// TIA Portal V17 export
// export: Created 2023-02-13T11:16:11.2408746Z, ExportSetting WithDefaults, DisplayName Totally Integrated Automation Portal, DisplayVersion V17, DisplayName TIA Portal Openness, DisplayVersion V17, DisplayName TIA Portal Teamcenter Gateway, DisplayVersion V17, DisplayName TIA Portal Version Control Interface, DisplayVersion V17, DisplayName SINAMICS Startdrive Advanced, DisplayVersion V17, DisplayName SINAMICS Startdrive G130, G150, S120, S150, SINAMICS MV, S210, DisplayVersion V17, DisplayName SINAMICS Startdrive G110M, G120, G120C, G120D, G120P, G115D, DisplayVersion V17, DisplayName STEP 7 Professional, DisplayVersion V17, DisplayName STEP 7 Safety, DisplayVersion V17, DisplayName WinCC Professional, DisplayVersion V17
DATA_BLOCK "Blend_T-31"   // DB214
VERSION : 0.1
// stored: AutoNumber false, DBAccessibleFromOPCUA true, DBAccessibleFromWebserver true, InstanceOfName Blend_Tank, InstanceOfType FB
"Blend_Tank"
   // VAR_INPUT
   //    IN_FBAV_Header1 : Bool;
   //    IN_FBAV_Header2 : Bool;
   //    IN_FBAV_Vinegar : Bool;
   //    IN_FBAV_Sugar : Bool;
   //    IN_FBAV_Salt : Bool;
   //    IN_FBAV_ProWater : Bool;
   //    IN_FBAV_Homomixer : Bool;
   //    IN_FBAV_Transfer1 : Bool;
   //    IN_FBAV_Transfer2 : Bool;
   //    IN_FBAV_Transfer3 : Bool;
   //    IN_FBAV_Outlet : Bool;
   //    IN_FBAV_CIP : Bool;
   //    IN_FBP_Transfer1 : Bool;
   //    IN_FBP_Transfer1_Sp : Real;
   //    IN_FBP_Transfer2 : Bool;
   //    IN_FBP_Transfer2_Sp : Real;
   //    IN_FBP_Transfer3 : Bool;
   //    IN_FBP_Transfer3_Sp : Real;
   //    IN_FBP_CIP : Bool;
   //    IN_FBP_CIP_Sp : Real;
   //    IN_LT01 : Real;
   //    "BFT-1 Prod Req" : Bool;
   //    "BFT-1 Prod Line" : Bool;
   //    "BFT-1 CIP Enable" : Bool;
   //    "BFT-1 CIPLine" : Bool;
   //    "BFT-2 Prod Req" : Bool;
   //    "BFT-2 Prod Line" : Bool;
   //    "BFT-2 CIP Enable" : Bool;
   //    "BFT-2 CIPLine" : Bool;
   //    "BFT-3 Prod Req" : Bool;
   //    "BFT-3 Prod Line" : Bool;
   //    "BFT-3 CIP Enable" : Bool;
   //    "BFT-3 CIPLine" : Bool;
   //    "Transfer 1 Busy" : Bool;
   //    "Transfer 2 Busy" : Bool;
   //    "Transfer 3 Busy" : Bool;
   //    "Header 1 Available" : Bool;
   //    "Header 2 Available" : Bool;
   //    "Vinegar Available" : Bool;
   //    "Sugar Available" : Bool;
   //    "Salt Available" : Bool;
   //    "ProWater Available" : Bool;
   //    "Homomixer Available" : Bool;
   //    IN_LDT : Date_And_Time;
   //    "CIP Pulse" : Bool;
   //    "CIP Supply ON" : Bool;
   //    "CIP Req OK" : Bool;
   //    "CIP Complete" : Bool;
   //    "CIP Busy" : Bool;
   // END_VAR
   // VAR_OUTPUT
   //    Out_AV_Header1 : Bool;
   //    Out_AV_Header2 : Bool;
   //    Out_AV_Vinegar : Bool;
   //    Out_AV_Sugar : Bool;
   //    Out_AV_Salt : Bool;
   //    Out_AV_ProWater : Bool;
   //    Out_AV_Homomixer : Bool;
   //    Out_AV_Transfer1 : Bool;
   //    Out_AV_Transfer2 : Bool;
   //    Out_AV_Transfer3 : Bool;
   //    Out_AV_Outlet : Bool;
   //    Out_AV_CIP : Bool;
   //    Out_P_Transfer1 : Bool;
   //    Out_P_Transfer1_Sp : Real;
   //    Out_P_Transfer2 : Bool;
   //    Out_P_Transfer2_Sp : Real;
   //    Out_P_Transfer3 : Bool;
   //    Out_P_Transfer3_Sp : Real;
   //    Out_P_CIP : Bool;
   //    Out_P_CIP_Sp : Real;
   //    Out_Agi : Bool;
   //    Out_Agi_Sp : Real;
   //    "Header 1 Req" : Bool;
   //    "Header 2 Req" : Bool;
   //    "Vinegar Req" : Bool;
   //    "Sugar Req" : Bool;
   //    "Salt Req" : Bool;
   //    "ProWater Req" : Bool;
   //    "Homomixer Req" : Bool;
   //    Out_CIP_Req : Bool;
   //    Out_CIP_Line_Open : Bool;
   // END_VAR
   // VAR
   //    Cmd : Struct
   //       "Ready For Transfer" : Bool;
   //       "CIP Tank 1" : Bool;
   //       "CIP Tank 2" : Bool;
   //       "CIP Line" : Bool;
   //       "Dose Head 1" : Bool;
   //       "Dose Head 2" : Bool;
   //       Agitator_Mode : Bool;
   //    END_STRUCT;
   // END_VAR
   // VAR RETAIN
   //    Param : Struct
   //       SP_Level_LL : Real;
   //       SP_Level_ML : Real;
   //       SP_Level_HL : Real;
   //       L_Hi_Lim : Real;
   //       L_Lo_Lim : Real;
   //       L_Hys : Real;
   //       LB_ON : Real;
   //       LB_OFF : Real;
   //       LB1_ON : Real;
   //       LB1_OFF : Real;
   //       LB2_ON : Real;
   //       LB2_OFF : Real;
   //       LB3_ON : Real;
   //       LB3_OFF : Real;
   //       SP_P1_Speed : Real;
   //       SP_P2_Speed : Real;
   //       SP_P3_Speed : Real;
   //       SP_LB_Speed : Real;
   //       SP_LB1_Speed : Real;
   //       SP_LB2_Speed : Real;
   //       SP_LB3_Speed : Real;
   //       CIP_Tank_P_Ret_Speed : Real;
   //       CIP_Ret_ON_SP : Real;
   //       CIP_Ret_OFF_SP : Real;
   //       Flushing_HW_Timer : Time;
   //    END_STRUCT;
   // END_VAR
   // VAR
   //    State : Struct
   //       "Tank LL" : Bool;
   //       "Tank ML" : Bool;
   //       "Tank HL" : Bool;
   //       LB_ON : Bool;
   //       LB1_ON : Bool;
   //       LB2_ON : Bool;
   //       LB3_ON : Bool;
   //       "CIP Tank" : Bool;
   //       "CIP Tank Ena" : Bool;
   //       "CIP Tank Ret 1 Ena" : Bool;
   //       "CIP Tank Ret 2 Ena" : Bool;
   //       "CIP Line" : Bool;
   //       "CIP Line Ena" : Bool;
   //       "CIP Return On" : Bool;
   //       "Dose On Prog" : Bool;
   //       "Dose EN" : Bool;
   //       "Ready For Transfer" : Bool;
   //       "Ready For Transfer Ena" : Bool;
   //       "BFT-1 EN" : Bool;
   //       "BFT-2 EN" : Bool;
   //       "BFT-3 EN" : Bool;
   //       "RM Dose" : Bool;
   //       "Transfer 1 On Progress" : Bool;
   //       "Transfer 2 On Progress" : Bool;
   //       "Transfer 3 On Progress" : Bool;
   //       "DoseHead1 ON" : Bool;
   //       "DoseHead2 ON" : Bool;
   //    END_STRUCT;
   //    Dose : Struct
   //       Dose_Start : DWord;
   //       Dose_Pause : DWord;
   //       Dose_Stop : DWord;
   //       Dose_State : DWord;
   //       Dose_Tank_Available : Word;
   //       Dose_Prod_Ready : Word;
   //       Dose_Header_Req : DWord;
   //       Dose_EN : Word;
   //    END_STRUCT;
   //    "Dose_Level_%" : Struct
   //       "ChiliAwetan1%" : Real;
   //       "ChiliAwetan2%" : Real;
   //       "ChiliAwetan3%" : Real;
   //       "Tomato%" : Real;
   //       "ChiliFresh1%" : Real;
   //       "ChiliFresh2%" : Real;
   //       "ChiliFresh3%" : Real;
   //       "Garlic%" : Real;
   //       "HW%" : Real;
   //       "Vinegar%" : Real;
   //       "Sugar%" : Real;
   //       "Salt%" : Real;
   //       "ProWater%" : Real;
   //       "Homomixer%" : Real;
   //    END_STRUCT;
   //    Dose_Level_Lit : Struct
   //       ChiliAwetan1Lit : Real;
   //       ChiliAwetan2Lit : Real;
   //       ChiliAwetan3Lit : Real;
   //       TomatoLit : Real;
   //       ChiliFresh1Lit : Real;
   //       ChiliFresh2Lit : Real;
   //       ChiliFresh3Lit : Real;
   //       GarlicLit : Real;
   //       HWLit : Real;
   //       VinegarLit : Real;
   //       SugarLit : Real;
   //       SaltLit : Real;
   //       ProWaterLit : Real;
   //       HomomixerLit : Real;
   //    END_STRUCT;
   //    SP_Dose_Level : Struct
   //       ChiliAwetan1Lit : Real;
   //       ChiliAwetan2Lit : Real;
   //       ChiliAwetan3Lit : Real;
   //       TomatoLit : Real;
   //       ChiliFresh1Lit : Real;
   //       ChiliFresh2Lit : Real;
   //       ChiliFresh3Lit : Real;
   //       GarlicLit : Real;
   //       HWLit : Real;
   //       VinegarLit : Real;
   //       SugarLit : Real;
   //       SaltLit : Real;
   //       ProWaterLit : Real;
   //       HomomixerLit : Real;
   //    END_STRUCT;
   //    r : Struct
   //       PosE1 : Bool;
   //       PosE2 : Bool;
   //       PosE3 : Bool;
   //       PosE4 : Bool;
   //       PosE5 : Bool;
   //       PosE6 : Bool;
   //       PosE7 : Bool;
   //       PosE8 : Bool;
   //       PosE9 : Bool;
   //       PosE10 : Bool;
   //       PosE11 : Bool;
   //       PosE12 : Bool;
   //       PosE13 : Bool;
   //       PosE14 : Bool;
   //       PosE15 : Bool;
   //       PosE16 : Bool;
   //       PosE17 : Bool;
   //       PosE18 : Bool;
   //       PosE19 : Bool;
   //       PosE20 : Bool;
   //       PosE21 : Bool;
   //       PosE22 : Bool;
   //       PosE23 : Bool;
   //       PosE24 : Bool;
   //       PosE25 : Bool;
   //       PosE26 : Bool;
   //       PosE27 : Bool;
   //       PosE28 : Bool;
   //       PosE29 : Bool;
   //       PosE30 : Bool;
   //       PosE31 : Bool;
   //       PosE32 : Bool;
   //    END_STRUCT;
   //    Actuator : Struct
   //       P_Transfer1 : Bool;
   //       P_Transfer2 : Bool;
   //       P_Transfer3 : Bool;
   //       AV_Transfer1 : Bool;
   //       AV_Transfer2 : Bool;
   //       AV_Transfer3 : Bool;
   //       AV_Outlet : Bool;
   //       AV_CIP_Tank : Bool;
   //    END_STRUCT;
   //    SP_ChiliAwetan1 : "RawDose";
   //    SP_ChiliAwetan2 : "RawDose";
   //    SP_ChiliAwetan3 : "RawDose";
   //    SP_Tomato : "RawDose";
   //    SP_ChiliFresh1 : "RawDose";
   //    SP_ChiliFresh2 : "RawDose";
   //    SP_ChiliFresh3 : "RawDose";
   //    SP_Garlic : "RawDose";
   //    SP_HW : "Raw_Pulse";
   //    SP_Vinegar : "RawDose";
   //    SP_Sugar : "RawDose";
   //    SP_Salt : "RawDose";
   //    SP_ProWater : "Raw_Pulse";
   //    SP_Homomixer : "RawDose";
   //    Dose_ChiliAwetan1 { S7_SetPoint := 'True'} : "DOSE";
   //    Dose_ChiliAwetan2 { S7_SetPoint := 'True'} : "DOSE";
   //    Dose_ChiliAwetan3 { S7_SetPoint := 'True'} : "DOSE";
   //    Dose_Tomato { S7_SetPoint := 'True'} : "DOSE";
   //    Dose_ChiliFresh1 { S7_SetPoint := 'True'} : "DOSE";
   //    Dose_ChiliFresh2 { S7_SetPoint := 'True'} : "DOSE";
   //    Dose_ChiliFresh3 { S7_SetPoint := 'True'} : "DOSE";
   //    Dose_Garlic { S7_SetPoint := 'True'} : "DOSE";
   //    Dose_HW { S7_SetPoint := 'True'} : "DOSE";
   //    Dose_Vinegar { S7_SetPoint := 'True'} : "DOSE";
   //    Dose_Sugar { S7_SetPoint := 'True'} : "DOSE";
   //    Dose_Salt { S7_SetPoint := 'True'} : "DOSE";
   //    Dose_ProWater { S7_SetPoint := 'True'} : "DOSE";
   //    Dose_Homomixer { S7_SetPoint := 'True'} : "DOSE";
   //    AlwaysON { S7_SetPoint := 'True'} : Bool;
   //    L_Hys_Abs { S7_SetPoint := 'True'} : Real;
   //    Hys_Level_HL : Real;
   //    Hys_Level_ML : Real;
   //    Hys_Level_LL : Real;
   //    TimerOff_Valve_Out : TON_TIME;
   //    TimerOff_Valve_P_1 { S7_SetPoint := 'True'} : TON_TIME;
   //    TimerOff_Valve_P_2 { S7_SetPoint := 'True'} : TON_TIME;
   //    TimerOff_Valve_P_3 { S7_SetPoint := 'True'} : TON_TIME;
   //    TimerOff_Valve_P_CIP { S7_SetPoint := 'True'} : TON_TIME;
   // END_VAR
   // VAR RETAIN
   //    Last_Dose_Qty : Struct
   //       ChiliAwetan1 : Real;
   //       ChiliAwetan2 : Real;
   //       ChiliAwetan3 : Real;
   //       Tomato : Real;
   //       ChiliFresh1 : Real;
   //       ChiliFresh2 : Real;
   //       ChiliFresh3 : Real;
   //       Garlic : Real;
   //       HW : Real;
   //       Vinegar : Real;
   //       Sugar : Real;
   //       Salt : Real;
   //       ProWater : Real;
   //       Homomixer : Real;
   //    END_STRUCT;
   // END_VAR
   // VAR
   //    "HW Flushing" : Struct
   //       Status : Struct
   //          "Flush to Blend" : Bool;
   //          "Flush to Drain" : Bool;
   //          Drain : Bool;
   //          Done : Bool;
   //       END_STRUCT;
   //       Qty : Struct
   //          "Flush to Blend Qty" : Real;
   //          "Flush to Drain Qty" : Real;
   //          "Flush to Blend Act" : Real;
   //          "Flush to Drain Act" : Real;
   //       END_STRUCT;
   //       TimeDrain_SP : DInt;
   //       Cmd_Start_Drain : Bool;
   //       Cmd_Stop_Drain : Bool;
   //       DrainTime : TONR_TIME;
   //    END_STRUCT;
   //    PumpTF1_OnDelay : TON_TIME;
   //    PumpTF2_OnDelay { S7_SetPoint := 'True'} : TON_TIME;
   //    PumpTF3_OnDelay { S7_SetPoint := 'True'} : TON_TIME;
   // END_VAR
   // VAR RETAIN
   //    TimerON : Struct
   //       TimerON_1 : TON_TIME;
   //       TimerON_2 { S7_SetPoint := 'True'} : TON_TIME;
   //       TimerON_3 { S7_SetPoint := 'True'} : TON_TIME;
   //       TimerON_4 { S7_SetPoint := 'True'} : TON_TIME;
   //       TimerON_5 { S7_SetPoint := 'True'} : TON_TIME;
   //       TimerON_6 { S7_SetPoint := 'True'} : TON_TIME;
   //       TimerON_7 { S7_SetPoint := 'True'} : TON_TIME;
   //       TimerON_8 { S7_SetPoint := 'True'} : TON_TIME;
   //    END_STRUCT;
   //    TimerOFF : Struct
   //       TimerOFF_1 : TOF_TIME;
   //       TimerOFF_2 { S7_SetPoint := 'True'} : TOF_TIME;
   //       TimerOFF_3 { S7_SetPoint := 'True'} : TOF_TIME;
   //       TimerOFF_4 { S7_SetPoint := 'True'} : TOF_TIME;
   //       TimerOFF_5 { S7_SetPoint := 'True'} : TOF_TIME;
   //       TimerOFF_6 { S7_SetPoint := 'True'} : TOF_TIME;
   //       TimerOFF_7 { S7_SetPoint := 'True'} : TOF_TIME;
   //       TimerOFF_8 { S7_SetPoint := 'True'} : TOF_TIME;
   //    END_STRUCT;
   // END_VAR
BEGIN
END_DATA_BLOCK
